FUNCTION_BLOCK SpecialDataWritingHandler
VAR_INPUT
	outletValveOpen : BOOL;
	saveActive : BOOL;
END_VAR
VAR_OUTPUT
	outletValveOpenArray : ARRAY[0..99] OF BOOL;
	outletValveOpenTimestamps : ARRAY[0..99] OF STRING;
	outletValveCloseArray : ARRAY[0..99] OF BOOL;
	outletValveCloseTimestamps : ARRAY[0..99] OF STRING;
END_VAR
VAR
	i : INT;
	specialDataSaveState : INT;
	openIndex : INT;
	closeIndex : INT;
	RTRIG_ValveOpened : R_TRIG;
	FTRIG_ValveClosed : F_TRIG;
	LocalTime     : FB_LocalSystemTime;
	currentOpenTime : DT;
	currentCloseTime : DT;
END_VAR


LocalTime(bEnable := TRUE);

CASE specialDataSaveState OF
	0:
	
		IF saveActive THEN
			specialDataSaveState := 1;
			resetDataArray();
		END_IF
	
	1:
		RTRIG_ValveOpened(CLK := outletValveOpen);
		FTRIG_ValveClosed(CLK := outletValveOpen);
		IF RTRIG_ValveOpened.Q THEN
			outletValveOpenArray[openIndex] := TRUE;
			currentOpenTime :=  SYSTEMTIME_TO_DT(LocalTime.systemTime);
			outletValveOpenTimestamps[openIndex] := CONCAT(CONCAT(TO_STRING(currentOpenTime),'.'),TO_STRING(LocalTime.systemTime.wMilliseconds));
			openIndex := openIndex + 1;
		END_IF
		IF FTRIG_ValveClosed.Q THEN
			outletValveCloseArray[closeIndex] := TRUE;
			currentCloseTime :=  SYSTEMTIME_TO_DT(LocalTime.systemTime);
			outletValveCloseTimeStamps[closeIndex] := CONCAT(CONCAT(TO_STRING(currentCloseTime),'.'),TO_STRING(LocalTime.systemTime.wMilliseconds));
			closeIndex := closeIndex + 1;
		END_IF
		
		IF NOT saveActive THEN
			openIndex := 0;
			closeIndex := 0;
			specialDataSaveState := 0;
		END_IF
	
END_CASE

METHOD resetDataArray : BOOL
VAR_INPUT
END_VAR

FOR i := 0 TO 99 DO
	outletValveOpenArray[i] := FALSE;
	outletValveOpenTimestamps[i] := '0';
	outletValveCloseArray[i] := FALSE;
	outletValveCloseTimestamps[i] := '0';
END_FOR
END_METHOD

END_FUNCTION_BLOCK

(* stored: Version 1.1.0.1, ProductVersion 3.1.4024.9
   POU SpecialDataWritingHandler: Id {c8b81348-d458-4793-8edc-72bcd9457d28}, SpecialFunc None
   Method resetDataArray: Id {84f98cca-f7b8-445f-b2e8-3768bad478a9} *)
